// TIA Portal V17 export
// export: Created 2023-02-14T02:49:13.0033818Z, ExportSetting WithDefaults, DisplayName Totally Integrated Automation Portal, DisplayVersion V17, DisplayName TIA Portal Openness, DisplayVersion V17, DisplayName TIA Portal Teamcenter Gateway, DisplayVersion V17, DisplayName TIA Portal Version Control Interface, DisplayVersion V17, DisplayName SINAMICS Startdrive Advanced, DisplayVersion V17, DisplayName SINAMICS Startdrive G130, G150, S120, S150, SINAMICS MV, S210, DisplayVersion V17, DisplayName SINAMICS Startdrive G110M, G120, G120C, G120D, G120P, G115D, DisplayVersion V17, DisplayName STEP 7 Professional, DisplayVersion V17, DisplayName STEP 7 Safety, DisplayVersion V17, DisplayName WinCC Professional, DisplayVersion V17
DATA_BLOCK "CIP_to_Mix"   // DB220
{ S7_Optimized_Access := 'FALSE' }
VERSION : 0.1
// stored: AutoNumber false, DBAccessibleFromOPCUA true, DBAccessibleFromWebserver true, IsOnlyStoredInLoadMemory false, IsWriteProtectedInAS false
   VAR
      HeartBeat : Bool := TRUE;
      CIP_RequestOK : Struct
         Header : Struct
            Header_CIP_RequestOK : Bool;
         END_STRUCT;
         "Chili Awetan" : Struct
            "T-02.00_CIP_RequestOK" : Bool;
            "T-03.00_CIP_RequestOK" : Bool;
            "T-04.00_CIP_RequestOK" : Bool;
         END_STRUCT;
         Tomato : Struct
            "T-05.00_CIP_RequestOK" : Bool;
         END_STRUCT;
         ChiliFresh : Struct
            "T-06.00_CIP_RequestOK" : Bool;
            "T-07.00_CIP_RequestOK" : Bool;
            "T-08.00_CIP_RequestOK" : Bool;
         END_STRUCT;
         Garlic : Struct
            "T-09.00_CIP_RequestOK" : Bool;
         END_STRUCT;
         Vinegar : Struct
            "T-10.00_CIP_RequestOK" : Bool;
         END_STRUCT;
         Homomixer : Struct
            "T-12.00_CIP_RequestOK" : Bool;
            "T-13.00_CIP_RequestOK" : Bool;
            "T-14.00_CIP_RequestOK" : Bool;
         END_STRUCT;
         "Blending Cluster 1" : Struct
            "T-20.00_CIP_RequestOK" : Bool;
            "T-21.00_CIP_RequestOK" : Bool;
            "T-30.00_CIP_RequestOK" : Bool;
            Blending_Cluster1_LineProduct_RequestOK : Bool;
            Free_CIP_RequestOK_1 : Bool;
            Free_CIP_RequestOK_2 : Bool;
         END_STRUCT;
         "Blending Cluster 2" : Struct
            "T-31.00_CIP_RequestOK" : Bool;
            "T-40.00_CIP_RequestOK" : Bool;
            "T-41.00_CIP_RequestOK" : Bool;
            Blending_Cluster2_LineProduct_RequestOK : Bool;
            Free_CIP_RequestOK_1 : Bool;
            Free_CIP_RequestOK_2 : Bool;
         END_STRUCT;
         "Rework Cluster 1" : Struct
            "T-22.00_CIP_RequestOK" : Bool;
         END_STRUCT;
         "Rework Cluster 2" : Struct
            "T-32.00_CIP_RequestOK" : Bool;
         END_STRUCT;
         "Buffer Cluster 1" : Struct
            "T-61.00_CIP_RequestOK" : Bool;
            "T-62.00_CIP_RequestOK" : Bool;
            "T61&T62_CIP_LineToPasteur_RequestOK" : Bool;
            "T-63.00_CIP_RequestOK" : Bool;
            "T-64.00_CIP_RequestOK" : Bool;
            "T63&T64_CIP_LineToPasteur_RequestOK" : Bool;
         END_STRUCT;
         "Buffer Cluster 2" : Struct
            "T-65.00_CIP_RequestOK" : Bool;
            "T-66.00_CIP_RequestOK" : Bool;
            "T65&T66_CIP_LineToPasteur_RequestOK" : Bool;
            "T-67.00_CIP_RequestOK" : Bool;
            "T-68.00_CIP_RequestOK" : Bool;
            "T67&T68_CIP_LineToPasteur_RequestOK" : Bool;
         END_STRUCT;
         "Storage THE 4" : Struct
            "T-23.00_CIP_RequestOK" : Bool;
            "T-24.00_CIP_RequestOK" : Bool;
            THE4_LineProduct_CIP_RequestOK : Bool;
         END_STRUCT;
         "Storage THE 5" : Struct
            "T-33.00_CIP_Tank_RequestOK" : Bool;
            "T-34.00_CIP_Tank_RequestOK" : Bool;
            "T33&T34_CIP_Line_RequestOK" : Bool;
            "T-35.00_CIP_Tank_RequestOK" : Bool;
            THE5_LineProduct_CIP_RequestOK : Bool;
         END_STRUCT;
         "T-79.00_CIP_RequestOK" : Bool;
         "T-81.00_CIP_RequestOK" : Bool;
         "T-84.00_CIP_RequestOK" : Bool;
         "T-85.00_CIP_RequestOK" : Bool;
         JBT_THE4_RequestOK : Bool;   // Open AV-22.11
         JBT_THE5_RequestOK : Bool;   // Open AV-22.11
         Aseptic_Pharmac_RequestOK : Bool;   // Open AV-39.06
         Free_CIP_RequestOK_8 : Bool;
         Free_CIP_RequestOK_9 : Bool;
         Free_CIP_RequestOK_10 : Bool;
         Free_CIP_RequestOK_11 : Bool;
         Free_CIP_RequestOK_12 : Bool;
         Free_CIP_RequestOK_13 : Bool;
         Free_CIP_RequestOK_14 : Bool;
         Free_CIP_RequestOK_15 : Bool;
         Free_CIP_RequestOK_16 : Bool;
         Osa_CIP_RequestOK : Bool;
         Free_CIP_RequestOK_18 : Bool;
         Free_CIP_RequestOK_19 : Bool;
         Free_CIP_RequestOK_20 : Bool;
         Free_CIP_RequestOK_21 : Bool;
         Free_CIP_RequestOK_22 : Bool;
         Free_CIP_RequestOK_23 : Bool;
         Free_CIP_RequestOK_24 : Bool;
      END_STRUCT;
      CIP_InProgress : Struct
         Header : Struct
            Header_CIP_InProgress : Bool;
         END_STRUCT;
         "Chili Awetan" : Struct
            "T-02.00_CIP_InProgress" : Bool;
            "T-03.00_CIP_InProgress" : Bool;
            "T-04.00_CIP_InProgress" : Bool;
         END_STRUCT;
         Tomato : Struct
            "T-05.00_CIP_InProgress" : Bool;
         END_STRUCT;
         ChiliFresh : Struct
            "T-06.00_CIP_InProgress" : Bool;
            "T-07.00_CIP_InProgress" : Bool;
            "T-08.00_CIP_InProgress" : Bool;
         END_STRUCT;
         Garlic : Struct
            "T-09.00_CIP_InProgress" : Bool;
         END_STRUCT;
         Vinegar : Struct
            "T-10.00_CIP_InProgress" : Bool;
         END_STRUCT;
         Homomixer : Struct
            "T-12.00_CIP_InProgress" : Bool;
            "T-13.00_CIP_InProgress" : Bool;
            "T-14.00_CIP_InProgress" : Bool;
         END_STRUCT;
         "Blending Cluster 1" : Struct
            "T-20.00_CIP_InProgress" : Bool;
            "T-21.00_CIP_InProgress" : Bool;
            "T-30.00_CIP_InProgress" : Bool;
            Blending_Cluster1_LineProduct_InProgress : Bool;
            Free_CIP_InProgress_1 : Bool;
            Free_CIP_InProgress_2 : Bool;
         END_STRUCT;
         "Blending Cluster 2" : Struct
            "T-31.00_CIP_InProgress" : Bool;
            "T-40.00_CIP_InProgress" : Bool;
            "T-41.00_CIP_InProgress" : Bool;
            Blending_Cluster2_LineProduct_InProgress : Bool;
            Free_CIP_InProgress_1 : Bool;
            Free_CIP_InProgress_2 : Bool;
         END_STRUCT;
         "Rework Cluster 1" : Struct
            "T-22.00_CIP_InProgress" : Bool;
         END_STRUCT;
         "Rework Cluster 2" : Struct
            "T-32.00_CIP_InProgress" : Bool;
         END_STRUCT;
         "Buffer Cluster 1" : Struct
            "T-61.00_CIP_InProgress" : Bool;
            "T-62.00_CIP_InProgress" : Bool;
            "T61&T62_CIP_LineToPasteur_InProgress" : Bool;
            "T-63.00_CIP_InProgress" : Bool;
            "T-64.00_CIP_InProgress" : Bool;
            "T63&T64_CIP_LineToPasteur_InProgress" : Bool;
         END_STRUCT;
         "Buffer Cluster 2" : Struct
            "T-65.00_CIP_InProgress" : Bool;
            "T-66.00_CIP_InProgress" : Bool;
            "T65&T66_CIP_LineToPasteur_InProgress" : Bool;
            "T-67.00_CIP_InProgress" : Bool;
            "T-68.00_CIP_InProgress" : Bool;
            "T67&T68_CIP_LineToPasteur_InProgress" : Bool;
         END_STRUCT;
         "Storage THE 4" : Struct
            "T-23.00_CIP_InProgress" : Bool;
            "T-24.00_CIP_InProgress" : Bool;
            THE4_LineProduct_CIP_InProgress : Bool;
         END_STRUCT;
         "Storage THE 5" : Struct
            "T-33.00_CIP_Tank_InProgress" : Bool;
            "T-34.00_CIP_Tank_InProgress" : Bool;
            "T33&T34_CIP_Line_InProgress" : Bool;
            "T-35.00_CIP_Tank_InProgress" : Bool;
            THE5_LineProduct_CIP_InProgress : Bool;
         END_STRUCT;
         "T-79.00_CIP_InProgress" : Bool;
         "T-81.00_CIP_InProgress" : Bool;
         "T-84.00_CIP_InProgress" : Bool;
         "T-85.00_CIP_InProgress" : Bool;
         Free_CIP_InProgress_5 : Bool;
         Free_CIP_InProgress_6 : Bool;
         Free_CIP_InProgress_7 : Bool;
         Free_CIP_InProgress_8 : Bool;
         Free_CIP_InProgress_9 : Bool;
         Free_CIP_InProgress_10 : Bool;
         Free_CIP_InProgress_11 : Bool;
         Free_CIP_InProgress_12 : Bool;
         Free_CIP_InProgress_13 : Bool;
         Free_CIP_InProgress_14 : Bool;
         Free_CIP_InProgress_15 : Bool;
         Free_CIP_InProgress_16 : Bool;
         Osa_CIP_InProgress : Bool;
         Free_CIP_InProgress_18 : Bool;
         Free_CIP_InProgress_19 : Bool;
         Free_CIP_InProgress_20 : Bool;
         Free_CIP_InProgress_21 : Bool;
         Free_CIP_InProgress_22 : Bool;
         Free_CIP_InProgress_23 : Bool;
         Free_CIP_InProgress_24 : Bool;
      END_STRUCT;
      CIP_Supply_On : Struct
         Header : Struct
            Header_CIP_Supply_ON : Bool;
         END_STRUCT;
         "Chili Awetan" : Struct
            "T-02.00_CIP_Supply_ON" : Bool;
            "T-03.00_CIP_Supply_ON" : Bool;
            "T-04.00_CIP_Supply_ON" : Bool;
         END_STRUCT;
         Tomato : Struct
            "T-05.00_CIP_Supply_ON" : Bool;
         END_STRUCT;
         ChiliFresh : Struct
            "T-06.00_CIP_Supply_ON" : Bool;
            "T-07.00_CIP_Supply_ON" : Bool;
            "T-08.00_CIP_Supply_ON" : Bool;
         END_STRUCT;
         Garlic : Struct
            "T-09.00_CIP_Supply_ON" : Bool;
         END_STRUCT;
         Vinegar : Struct
            "T-10.00_CIP_Supply_ON" : Bool;
         END_STRUCT;
         Homomixer : Struct
            "T-12.00_CIP_Supply_ON" : Bool;
            "T-13.00_CIP_Supply_ON" : Bool;
            "T-14.00_CIP_Supply_ON" : Bool;
         END_STRUCT;
         "Blending Cluster 1" : Struct
            "T-20.00_CIP_Supply_ON" : Bool;
            "T-21.00_CIP_Supply_ON" : Bool;
            "T-30.00_CIP_Supply_ON" : Bool;
            Blending_Cluster1_LineProduct_Supply_ON : Bool;
            Free_CIP_Supply_ON_1 : Bool;
            Free_CIP_Supply_ON_2 : Bool;
         END_STRUCT;
         "Blending Cluster 2" : Struct
            "T-31.00_CIP_Supply_ON" : Bool;
            "T-40.00_CIP_Supply_ON" : Bool;
            "T-41.00_CIP_Supply_ON" : Bool;
            Blending_Cluster2_LineProduct_Supply_ON : Bool;
            Free_CIP_Supply_ON_1 : Bool;
            Free_CIP_Supply_ON_2 : Bool;
         END_STRUCT;
         "Rework Cluster 1" : Struct
            "T-22.00_CIP_Supply_ON" : Bool;
         END_STRUCT;
         "Rework Cluster 2" : Struct
            "T-32.00_CIP_Supply_ON" : Bool;
         END_STRUCT;
         "Buffer Cluster 1" : Struct
            "T-61.00_CIP_Supply_ON" : Bool;
            "T-62.00_CIP_Supply_ON" : Bool;
            "T61&T62_CIP_LineToPasteur_Supply_ON" : Bool;
            "T-63.00_CIP_Supply_ON" : Bool;
            "T-64.00_CIP_Supply_ON" : Bool;
            "T63&T64_CIP_LineToPasteur_Supply_ON" : Bool;
         END_STRUCT;
         "Buffer Cluster 2" : Struct
            "T-65.00_CIP_Supply_ON" : Bool;
            "T-66.00_CIP_Supply_ON" : Bool;
            "T65&T66_CIP_LineToPasteur_Supply_ON" : Bool;
            "T-67.00_CIP_Supply_ON" : Bool;
            "T-68.00_CIP_Supply_ON" : Bool;
            "T67&T68_CIP_LineToPasteur_Supply_ON" : Bool;
         END_STRUCT;
         "Storage THE 4" : Struct
            "T-23.00_CIP_Supply_ON" : Bool;
            "T-24.00_CIP_Supply_ON" : Bool;
            THE4_LineProduct_CIP_Supply_ON : Bool;
         END_STRUCT;
         "Storage THE 5" : Struct
            "T-33.00_CIP_Tank_Supply_ON" : Bool;
            "T-34.00_CIP_Tank_Supply_ON" : Bool;
            "T33&T34_CIP_Line_Supply_ON" : Bool;
            "T-35.00_CIP_Tank_Supply_ON" : Bool;
            THE5_LineProduct_CIP_Supply_ON : Bool;
         END_STRUCT;
         "T-79.00_CIP_Supply_ON" : Bool;
         "T-81.00_CIP_Supply_ON" : Bool;
         "T-84.00_CIP_Supply_ON" : Bool;
         "T-85.00_CIP_Supply_ON" : Bool;
         Free_CIP_Supply_ON_5 : Bool;
         Free_CIP_Supply_ON_6 : Bool;
         Free_CIP_Supply_ON_7 : Bool;
         Free_CIP_Supply_ON_8 : Bool;
         Free_CIP_Supply_ON_9 : Bool;
         Free_CIP_Supply_ON_10 : Bool;
         Free_CIP_Supply_ON_11 : Bool;
         Free_CIP_Supply_ON_12 : Bool;
         Free_CIP_Supply_ON_13 : Bool;
         Free_CIP_Supply_ON_14 : Bool;
         Free_CIP_Supply_ON_15 : Bool;
         Free_CIP_Supply_ON_16 : Bool;
         Osa_CIP_Supply_ON : Bool;
         Free_CIP_Supply_ON_18 : Bool;
         Free_CIP_Supply_ON_19 : Bool;
         Free_CIP_Supply_ON_20 : Bool;
         Free_CIP_Supply_ON_21 : Bool;
         Free_CIP_Supply_ON_22 : Bool;
         Free_CIP_Supply_ON_23 : Bool;
         Free_CIP_Supply_ON_24 : Bool;
      END_STRUCT;
      CIP_Complete : Struct
         Header : Struct
            Header_CIP_Complete : Bool;
         END_STRUCT;
         "Chili Awetan" : Struct
            "T-02.00_CIP_Complete" : Bool;
            "T-03.00_CIP_Complete" : Bool;
            "T-04.00_CIP_Complete" : Bool;
         END_STRUCT;
         Tomato : Struct
            "T-05.00_CIP_Complete" : Bool;
         END_STRUCT;
         ChiliFresh : Struct
            "T-06.00_CIP_Complete" : Bool;
            "T-07.00_CIP_Complete" : Bool;
            "T-08.00_CIP_Complete" : Bool;
         END_STRUCT;
         Garlic : Struct
            "T-09.00_CIP_Complete" : Bool;
         END_STRUCT;
         Vinegar : Struct
            "T-10.00_CIP_Complete" : Bool;
         END_STRUCT;
         Homomixer : Struct
            "T-12.00_CIP_Complete" : Bool;
            "T-13.00_CIP_Complete" : Bool;
            "T-14.00_CIP_Complete" : Bool;
         END_STRUCT;
         "Blending Cluster 1" : Struct
            "T-20.00_CIP_Complete" : Bool;
            "T-21.00_CIP_Complete" : Bool;
            "T-30.00_CIP_Complete" : Bool;
            Blending_Cluster1_LineProduct_Complete : Bool;
            Free_CIP_Complete_1 : Bool;
            Free_CIP_Complete_2 : Bool;
         END_STRUCT;
         "Blending Cluster 2" : Struct
            "T-31.00_CIP_Complete" : Bool;
            "T-40.00_CIP_Complete" : Bool;
            "T-41.00_CIP_Complete" : Bool;
            Blending_Cluster2_LineProduct_Complete : Bool;
            Free_CIP_Complete_1 : Bool;
            Free_CIP_Complete_2 : Bool;
         END_STRUCT;
         "Rework Cluster 1" : Struct
            "T-22.00_CIP_Complete" : Bool;
         END_STRUCT;
         "Rework Cluster 2" : Struct
            "T-32.00_CIP_Complete" : Bool;
         END_STRUCT;
         "Buffer Cluster 1" : Struct
            "T-61.00_CIP_Complete" : Bool;
            "T-62.00_CIP_Complete" : Bool;
            "T61&T62_CIP_LineToPasteur_Complete" : Bool;
            "T-63.00_CIP_Complete" : Bool;
            "T-64.00_CIP_Complete" : Bool;
            "T63&T64_CIP_LineToPasteur_Complete" : Bool;
         END_STRUCT;
         "Buffer Cluster 2" : Struct
            "T-65.00_CIP_Complete" : Bool;
            "T-66.00_CIP_Complete" : Bool;
            "T65&T66_CIP_LineToPasteur_Complete" : Bool;
            "T-67.00_CIP_Complete" : Bool;
            "T-68.00_CIP_Complete" : Bool;
            "T67&T68_CIP_LineToPasteur_Complete" : Bool;
         END_STRUCT;
         "Storage THE 4" : Struct
            "T-23.00_CIP_Complete" : Bool;
            "T-24.00_CIP_Complete" : Bool;
            THE4_LineProduct_CIP_Complete : Bool;
         END_STRUCT;
         "Storage THE 5" : Struct
            "T-33.00_CIP_Tank_Complete" : Bool;
            "T-34.00_CIP_Tank_Complete" : Bool;
            "T33&T34_CIP_Line_Complete" : Bool;
            "T-35.00_CIP_Tank_Complete" : Bool;
            THE5_LineProduct_CIP_Complete : Bool;
         END_STRUCT;
         "T-79.00_CIP_Complete" : Bool;
         "T-81.00_CIP_Complete" : Bool;
         "T-84.00_CIP_Complete" : Bool;
         "T-85.00_CIP_Complete" : Bool;
         Free_CIP_Complete_5 : Bool;
         Free_CIP_Complete_6 : Bool;
         Free_CIP_Complete_7 : Bool;
         Free_CIP_Complete_8 : Bool;
         Free_CIP_Complete_9 : Bool;
         Free_CIP_Complete_10 : Bool;
         Free_CIP_Complete_11 : Bool;
         Free_CIP_Complete_12 : Bool;
         Free_CIP_Complete_13 : Bool;
         Free_CIP_Complete_14 : Bool;
         Free_CIP_Complete_15 : Bool;
         Free_CIP_Complete_16 : Bool;
         Osa_CIP_Complete : Bool;
         Free_CIP_Complete_18 : Bool;
         Free_CIP_Complete_19 : Bool;
         Free_CIP_Complete_20 : Bool;
         Free_CIP_Complete_21 : Bool;
         Free_CIP_Complete_22 : Bool;
         Free_CIP_Complete_23 : Bool;
         Free_CIP_Complete_24 : Bool;
      END_STRUCT;
   END_VAR
BEGIN
END_DATA_BLOCK
